TYPE ST_TCPConnection_HMI_CMD :
STRUCT
	bWriteSocketConnect		:BOOL;
	bReadSocketConnect		:BOOL;
	bResetRegistry			:BOOL;
END_STRUCT
END_TYPE

(* stored: Version 1.1.0.1, ProductVersion 3.1.4024.12
   DUT ST_TCPConnection_HMI_CMD: Id {84b01e7f-4d40-40b0-aab8-df3f6dbbd392} *)
